FUNCTION_BLOCK ABSTRACT FB_CylinderBase EXTENDS FB_ComponentBase IMPLEMENTS ITF_CylinderBase		//Abstract (non-instantiable) base definition from which numerous varieties of Cylinders may be derived through function block extension.
VAR_INPUT
END_VAR
VAR_OUTPUT
END_VAR
VAR CONSTANT
	//Constant declarations
	CYLINDER_BASE_ALARM_COUNT	: UDINT := 16;
END_VAR
VAR
	//ITF_Cylinder internal property variables
	tExtendTime		: TIME := T#1S;		//Approximate expected time for the cylinder to complete an extension cycle
	tRetractTime 	: TIME := T#1S;		//Approximate expected time for the cylinder to complete a retraction cycle
	fTimeoutFactor	: LREAL := 1.5;		//Multiplicative factor that determines error timeout threshold based on the expected cycle time
	bExtended 		: BOOL;				//Status bit for the position of the cylinder
	bRetracted		: BOOL;				//Status bit for the position of the cylinder
	bExtending		: BOOL;				//Cylinder is currently extending
	bRetracting		: BOOL;				//Cylinder is currently retracting
	bExtendOutput	: BOOL;				//Cylinder "extend" output is currently active
	bRetractOutput	: BOOL; 			//Cylinder "retract" output is currently active

	//Alarming
	a_fbCylinderBaseAlarms : ARRAY[1..CYLINDER_BASE_ALARM_COUNT] OF FB_TcAlarm;
	
	//HMI monitoring and control structure
	stCylinderBaseHMI		: ST_CylinderBase_HMI;
	
	//Internal Variables
	fbExtensionTimeout_TON		: Tc2_Standard.TON;		//Timer for monitoring extension timeouts
	tExtensionTimeout			: TIME;					//Extension timeout threshold calculated from expected ExtendTime and TimeoutFactor
	fbRetractionTimeout_TON		: Tc2_Standard.TON;		//Timer for monitoring retraction timeouts
	tRetractionTimeout			: TIME;					//Retraction timeout threshold calculated from expected RetractTime and TimeoutFactor
	bExtendRequest				: BOOL;					//Extension request received
	bRetractRequest				: BOOL;					//Retraction request received
	bExtendCommand				: BOOL;					//Direct command to be sent to outputs
	bRetractCommand				: BOOL;					//Direct command to be sent to outputs
	bExtendedFeedback			: BOOL;					//Direct feedback value from inputs
	bRetractedFeedback			: BOOL;					//Direct feedback value from inputs
	bIncomingRequest			: BOOL;					//New external request has been made
	
	
	//Simulation variables
	fbSimExtend_TON		: Tc2_Standard.TON;
	fbSimRetract_TON	: Tc2_Standard.TON;
	bSimExtendCommand	: BOOL;
	bSimRetractCommand	: BOOL;
END_VAR

METHOD ErrorOperation : BOOL
VAR_INPUT
END_VAR
bExtendCommand := FALSE;
bRetractCommand := FALSE;
END_METHOD

METHOD Extend : BOOL
bExtendRequest := TRUE;
bRetractRequest := FALSE;
bIncomingRequest := TRUE;
END_METHOD

PROPERTY Extended : BOOL	//Status bit for the position of the cylinder
GET
Extended := bExtended;
END_GET
END_PROPERTY

PROPERTY Extending : BOOL
GET
Extending := bExtending;
END_GET
END_PROPERTY

PROPERTY ExtendOutput : BOOL
GET
ExtendOutput := bExtendOutput;
END_GET
END_PROPERTY

PROPERTY ExtendTime : TIME	//Approximate expected time for the cylinder to complete an extension cycle
GET
ExtendTime := tExtendTime;
END_GET
SET
tExtendTime := ExtendTime;
END_SET
END_PROPERTY

METHOD HMICommunication : BOOL
SUPER^.HMICommunication();		//Call the base method

//Process HMI requests
IF stCylinderBaseHMI.bIncomingHMIRequest AND NOT stCylinderBaseHMI.bHMICommandConfirmation THEN		//If a request has been issued by the HMI, and a previous request has not just finished being processed
	IF stCylinderBaseHMI.bHMIControlAvailable THEN		//If the current conditions permit HMI control (Should be determined by the extended application components)
		IF stCylinderBaseHMI.bExtendHMIRequest THEN		//Execute the active requests
			Extend();
			stCylinderBaseHMI.bHMICommandConfirmation := TRUE;	//Confirm that the request has been processed
		END_IF
		IF stCylinderBaseHMI.bRetractHMIRequest THEN
			Retract();
			stCylinderBaseHMI.bHMICommandConfirmation := TRUE;	//Confirm that the request has been processed
		END_IF
		IF stCylinderBaseHMI.bIdleHMIRequest THEN
			Idle();
			stCylinderBaseHMI.bHMICommandConfirmation := TRUE;	//Confirm that the request has been processed
		END_IF
		IF stCylinderBaseHMI.bExtendTimeHMISetRequest THEN
			ExtendTime := stCylinderBaseHMI.tExtendTimeHMISetValue;
			stCylinderBaseHMI.bHMICommandConfirmation := TRUE;	//Confirm that the request has been processed
		END_IF
		IF stCylinderBaseHMI.bRetractTimeHMISetRequest THEN
			RetractTime := stCylinderBaseHMI.tRetractTimeHMISetValue;
			stCylinderBaseHMI.bHMICommandConfirmation := TRUE;	//Confirm that the request has been processed
		END_IF
		IF stCylinderBaseHMI.bTimeoutFactorHMISetRequest THEN
			TimeoutFactor := stCylinderBaseHMI.fTimeoutFactorHMISetValue;
			stCylinderBaseHMI.bHMICommandConfirmation := TRUE;	//Confirm that the request has been processed
		END_IF
	END_IF
END_IF


//Update HMI status info
stCylinderBaseHMI.tExtendTime := tExtendTime;
stCylinderBaseHMI.tRetractTime := tRetractTime;
stCylinderBaseHMI.fTimeoutFactor := fTimeoutFactor;
stCylinderBaseHMI.bExtended := bExtended;
stCylinderBaseHMI.bExtending := bExtending;
stCylinderBaseHMI.bRetracted := bRetracted;
stCylinderBaseHMI.bRetracting := bRetracting;
stCylinderBaseHMI.bExtendCommand := bExtendCommand OR bSimExtendCommand;
stCylinderBaseHMI.bRetractCommand := bRetractCommand OR bSimRetractCommand;
END_METHOD

METHOD Idle : BOOL
bExtendRequest := FALSE;
bRetractRequest := FALSE;
bIncomingRequest := TRUE;
END_METHOD

METHOD initialize : BOOL
VAR_INPUT
END_VAR

VAR
	sTemp: STRING;
END_VAR
SUPER^.initialize();

sTemp := CONCAT(CONCAT(CONCAT('Cylinder ', ': '), sName), ' '); 	//Creates a utility string for alarms and other messaging that reads (example text) - "Module 10 - Main Casepacker" to be followed by the alarm or message info
//TODO: Rename Event Class to AxisBase
F_CreateAllEventsInClass(	p_aAlarms := a_fbCylinderBaseAlarms,
							nClassSize := SIZEOF(TC_EVENTS.CylinderBase),
							pInitEvent := ADR(TC_EVENTS.CylinderBase.InitReferenceEvent),
							sPrefix := sTemp );
END_METHOD

METHOD Monitoring : BOOL
VAR_INPUT
END_VAR
SUPER^.Monitoring();

IF NOT bError THEN
	tExtensionTimeout := LREAL_TO_TIME(TIME_TO_LREAL(tExtendTime) * fTimeoutFactor);
	tRetractionTimeout := LREAL_TO_TIME(TIME_TO_LREAL(tRetractTime) * fTimeoutFactor);
	
	fbExtensionTimeout_TON(IN := bExtending, PT := tExtensionTimeout);	//Timer for monitoring extension timeout, PT = Extension time multiplied by the timeout factor
	fbRetractionTimeout_TON(IN := bRetracting, PT := tRetractionTimeout);	//Timer for monitoring retraction timeout, PT = Retraction time multiplied by the timeout factor

	//Simultaneous extend and retract commands throw an invalid command error
	IF 		(bExtending AND bRetracting)
		OR 	(bExtendRequest AND bRetractRequest)
		OR 	(bExtendCommand AND bRetractCommand) THEN 
		nErrorID := E_CylinderBase.InvalidCommand;
	END_IF
	
	//If both extended and retracted feedback are true at any point, throw an invalid position error
	IF bExtended AND bRetracted THEN
		bError := TRUE;
		nErrorID := E_CylinderBase.InvalidPositionStatus;
	END_IF
	
	//If the cylinder takes longer than expected to extend, throw a timeout error
	IF fbExtensionTimeout_TON.Q THEN
		bError := TRUE;
		nErrorID := E_CylinderBase.ExtendTimeout;
	END_IF
	
	//If the cylinder takes longer than expected to retract, throw a timeout error
	IF fbRetractionTimeout_TON.Q THEN
		bError := TRUE;
		nErrorID := E_CylinderBase.RetractTimeout;
	END_IF
END_IF

//If cylinder is in motion toward a position, but it has not yet been reached, set busy bit
IF (bExtending) OR (bRetracting) THEN
	bActive := TRUE;
ELSE
	bActive := FALSE;
END_IF

IF bSimExtendCommand OR bExtendCommand THEN
	bExtendOutput := TRUE;
ELSE
	bExtendOutput := FALSE;
END_IF

IF bSimRetractCommand OR bRetractCommand THEN
	bRetractOutput := TRUE;
ELSE
	bRetractOutput := FALSE;
END_IF
END_METHOD

METHOD Reset : BOOL
SUPER^.Reset();

bExtending := FALSE;
bRetracting := FALSE;

fbSimExtend_TON.IN := FALSE;
fbSimRetract_TON.IN := FALSE;

bExtendCommand := FALSE;
bRetractCommand := FALSE;
END_METHOD

METHOD Retract : UDINT
bRetractRequest := TRUE;
bExtendRequest := FALSE;
bIncomingRequest := TRUE;
END_METHOD

PROPERTY Retracted : BOOL	//Status bit for the position of the cylinder
GET
Retracted := bRetracted;
END_GET
END_PROPERTY

PROPERTY Retracting : BOOL
GET
Retracting := bRetracting;
END_GET
END_PROPERTY

PROPERTY RetractOutput : BOOL
GET
RetractOutput := bRetractOutput;
END_GET
END_PROPERTY

PROPERTY RetractTime : TIME
GET
RetractTime := tRetractTime;
END_GET
SET
tRetractTime := RetractTime;
END_SET
END_PROPERTY

METHOD SimulateOperation : BOOL
VAR_INPUT
END_VAR
IF bEnabled THEN
	
	bExtendCommand := FALSE;		//Hardware commands should be disabled during simulation mode
	bRetractCommand := FALSE;		//Hardware commands should be disabled during simulation mode
	
	fbSimExtend_TON();		//Call timer FB
	fbSimRetract_TON();		//Call timer FB
	
	IF fbSimExtend_TON.Q THEN		//Whenever the extend timer completes, set status to extended and turn off the timer
		bExtended := TRUE;
		fbSimExtend_TON.IN := FALSE;
	END_IF
	
	IF fbSimRetract_TON.Q THEN		//Whenever the retract timer completes, set status to retracted and turn off the timer
		bRetracted := TRUE;
		fbSimRetract_TON.IN := FALSE;
	END_IF
	
	IF bIncomingRequest THEN
		IF bExtendRequest THEN					//Whenever a new extend request comes in, check to see if we are still currently timing a retract action
			IF fbSimRetract_TON.IN THEN			//If a retract action is still in progress, appropriately scale the extend time to account for the distance traveled during the in-process retraction
				fbSimExtend_TON.PT := tExtendTime * (TIME_TO_UDINT(fbSimRetract_TON.ET) / TIME_TO_UDINT(tRetractTime));		//partial extend time = (full distance extend time) * (proportional distance covered during retraction)
				bSimRetractCommand := FALSE;
				fbSimRetract_TON.IN := FALSE;	//Disable retract timer
			ELSE
				fbSimExtend_TON.PT := tExtendTime;	//If no retraction was active, assume we are currently at fully retracted position, or this is the first command the cylinder has received, so initialize to full extend time
			END_IF
			bRetracted := FALSE;
			bSimRetractCommand := FALSE;
			bSimExtendCommand := TRUE;
			fbSimExtend_TON.IN := TRUE;				//Activate the extension timer
		ELSIF bRetractRequest THEN					//Same as above, but reversed
			IF fbSimExtend_TON.IN THEN
				fbSimRetract_TON.PT := tRetractTime * (TIME_TO_UDINT(fbSimExtend_TON.ET) / TIME_TO_UDINT(tRetractTime));
				bSimExtendCommand := FALSE;
				fbSimExtend_TON.IN := FALSE;
			ELSE
				fbSimRetract_TON.PT := tRetractTime;
			END_IF
			bExtended := FALSE;
			fbSimRetract_TON.IN := TRUE;
			bSimExtendCommand := FALSE;
			bSimRetractCommand := TRUE;
		ELSE
			bExtended := FALSE;
			bRetracted := FALSE;
			
			fbSimExtend_TON.IN := FALSE;			
			fbSimRetract_TON.IN := FALSE;
			
			bSimExtendCommand := FALSE;
			bSimRetractCommand := FALSE;
		END_IF
		bIncomingRequest := FALSE;
	END_IF
	
	bExtending := fbSimExtend_TON.IN;
	bRetracting := fbSimRetract_TON.IN;
ELSE
	bIncomingRequest := FALSE;
	fbSimExtend_TON.IN := FALSE;
	fbSimRetract_TON.IN := FALSE;
END_IF
END_METHOD

METHOD StandardOperation : BOOL
VAR_INPUT
END_VAR
IF bEnabled THEN
	IF bIncomingRequest THEN
		bExtendCommand := bExtendRequest;
		bRetractCommand := bRetractRequest;
		bIncomingRequest := FALSE;
	END_IF
	
	IF bExtendCommand AND NOT bExtended THEN
		bExtending := TRUE;
	END_IF
	
	IF bRetractCommand AND NOT bRetracted THEN
		bRetracting := TRUE;
	END_IF
	
	bExtended := bExtendedFeedback;
	bRetracted := bRetractedFeedback;
ELSE
	bIncomingRequest := FALSE;
END_IF
END_METHOD

PROPERTY TimeoutFactor : LREAL	//Multiplicative factor that determines error timeout threshold based on the expected time
GET
TimeoutFactor := fTimeoutFactor;
END_GET
SET
fTimeoutFactor := TimeoutFactor;
END_SET
END_PROPERTY

END_FUNCTION_BLOCK

(* stored: Version 1.1.0.1, ProductVersion 3.1.4024.9
   POU FB_CylinderBase: Id {52da9de5-3fad-4063-acc0-baf4f434d3da}, SpecialFunc None
   Folder 01_SUPER_Overrides: Id {3759e4fb-4932-4bdf-a384-c91488a99c06}
   Folder 02_ITF_CylinderBase: Id {fd62914a-ce7f-45e1-a60f-6b0a8f056fa6}
   Folder 01_Properties: Id {8e42ea4e-7181-4c37-8410-860072bf559d}
   Folder 01_Config: Id {55fa993a-c06b-4028-b1a7-5143879c9882}
   Folder 02_Control: Id {ccee1f0d-4c1d-4948-be0b-d67086a5625a}
   Folder 03_Status: Id {a6c30b2c-9909-4495-9112-fe04e1710960}
   Folder 02_Methods: Id {134e066b-1864-45a9-b950-def6585b175a}
   Method ErrorOperation: Id {8d55c932-b7f7-4c17-b6cb-b28020145d63}
   Method Extend: Id {f2f50916-95c8-4296-81fa-2eb45fed1456}
   Property Extended: Id {128445b1-3e80-4708-b9e1-19ce6b51555e}
   Get Get: Id {781ffbcf-f0dd-4cfe-9ab3-9d16fba8d804}
   Property Extending: Id {8dc2b23f-dc4a-4aaf-9b9e-4760571c2eff}
   Get Get: Id {b2a18490-80bd-4781-9d86-ccc9598925b0}
   Property ExtendOutput: Id {a07bfd4f-6440-40b8-8c6f-596e6b612958}
   Get Get: Id {b9d9d74a-1032-4e17-acbc-35de9f9613d9}
   Property ExtendTime: Id {a4075211-1976-400b-8eea-c3bc8ac07233}
   Get Get: Id {e59f7847-22d0-41fe-998f-efe63fb99e79}
   Set Set: Id {f413e2a7-c6ea-46a9-8129-6cd42817fadf}
   Method HMICommunication: Id {53a5999d-4f0f-49ef-ab47-409900876100}
   Method Idle: Id {6860462f-376a-4f39-8e43-cc88a6e1061d}
   Method initialize: Id {fb290f3c-3753-4f5a-a80b-69d733f51e19}
   Method Monitoring: Id {1b05306f-5859-4831-8fa0-dfd8904003bf}
   Method Reset: Id {2939002c-4b5f-4b1b-957e-dc41265429f6}
   Method Retract: Id {ddd5b4d4-6775-4df5-94dc-a4f52cd08d94}
   Property Retracted: Id {68547752-56e1-4d64-a9dd-3a591e9a96e3}
   Get Get: Id {b42bac66-19df-48df-b3cc-977f073a754f}
   Property Retracting: Id {84a5612f-2482-4d3b-a71e-8122965942f4}
   Get Get: Id {9078e90f-4f2f-4f58-94da-32decfc9b92e}
   Property RetractOutput: Id {45884ba1-8eec-4095-9faf-e3d1372e359b}
   Get Get: Id {c23c6549-2e8b-4a28-a67a-38ec8e737af3}
   Property RetractTime: Id {f7614a09-0bff-4962-9883-4ae606194bce}
   Get Get: Id {55693881-357c-432d-85c1-e641c9d1be69}
   Set Set: Id {14fd22a6-6df7-490a-84c4-56417826ff85}
   Method SimulateOperation: Id {7b675cac-d1b5-41ff-8c29-f3ee23a7c4f2}
   Method StandardOperation: Id {5b749516-6da3-4cb2-b6d8-1ea76986585c}
   Property TimeoutFactor: Id {149cf3c6-73fd-4da9-8764-afb5280fce49}
   Get Get: Id {8cdb479a-6c81-42b4-8c38-f64e2bdbbd37}
   Set Set: Id {bd408ab2-e9a1-4e87-be5e-ba8cd910121d} *)
